// TIA Portal project "1200_SQL" (V16)

(* hardware
DEVICE "S7-1200 station_1"  S7-1200 Station
   slot 0: "Rack_0"  S7-1200 Rack  Rack  V1.0
   slot 1: "PLC_1"  CPU 1215C DC/DC/Rly  6ES7 215-1HG40-0XB0  V4.4
*)

// ===== PLC "PLC_1"  CPU 1215C DC/DC/Rly =====

VAR_GLOBAL   // PLC tag table "Default tag table"
   "Tag_1" AT %M10.0 : Bool;
   "Tag_2" AT %M30.0 : Bool;
   "System_Byte" AT %MB1 : Byte;
   "FirstScan" AT %M1.0 : Bool;
   "DiagStatusUpdate" AT %M1.1 : Bool;
   "AlwaysTRUE" AT %M1.2 : Bool;
   "AlwaysFALSE" AT %M1.3 : Bool;
   "Clock_Byte" AT %MB0 : Byte;
   "Clock_10Hz" AT %M0.0 : Bool;
   "Clock_5Hz" AT %M0.1 : Bool;
   "Clock_2.5Hz" AT %M0.2 : Bool;
   "Clock_2Hz" AT %M0.3 : Bool;
   "Clock_1.25Hz" AT %M0.4 : Bool;
   "Clock_1Hz" AT %M0.5 : Bool;
   "Clock_0.625Hz" AT %M0.6 : Bool;
   "Clock_0.5Hz" AT %M0.7 : Bool;
   "Tag_3" AT %M1000.0 : Bool;
   "Tag_4" AT %M1000.1 : Bool;
   "Tag_5" AT %M1000.2 : Bool;
   "Tag_6" AT %M29.0 : Bool;
   "Tag_7" AT %M1000.5 : Bool;
END_VAR

TYPE "typeUseCaseSpecificTokenRow"
   STRUCT
      length : Byte;
      data : DWord;
   END_STRUCT;
END_TYPE

TYPE "typeUseCaseSpecificData"
   STRUCT
      header : "LSql_typeTDSPacketHeader";   // TDS Protocol header
      tokenColumnMetaData : Array[0..23] of Byte;   // information about the columns returned in the tokenRows - depends on user data
      tokenRows : Array[0..14] of "typeUseCaseSpecificTokenRow";   // Rows returned for the SQL Batch - sturcture depends on user data!
      bytes : Array[0..867] of Byte;
   END_STRUCT;
   // // header."type" : type of TDS package (4 = Server Response)
   // // header.status : status of the TDS package (1= last package, 0 = more packages follow)
   // // header.length : length of the TDS response
   // // header.SPID : process id of the SQL server
   // // header.PacketID : id of one message for a paket
   // // header.Window : not used - should be ignored by user
END_TYPE

// folder: LSql

TYPE "LSql_typeDiagnostics"
TITLE = typeDiagnosticsTemplate
   STRUCT
      status : Word;   // Status of the Block or error identification when error occurred
      subfunctionStatus : Word;   // Status or return value of called FB's, FCs and system blocks
      stateNumber : DInt;   // State in the state machine of the block where the error occurred
   END_STRUCT;
END_TYPE

TYPE "LSql_typeLoginInformation"
   STRUCT
      hostName : String;   // optional: name of local host
      userName : String;   // mandatory: username for login to database
      password : String;   // mandatory: password for login to database
      appName : String;   // optional: name of app connectiong to database
      serverName : String;   // mandatory: servername of database
      libraryName : String;   // optional: name of ui
      local : String;   // optional: language used in ui
      databaseName : String;   // mandatory: database to read or write from
      sspi : String;   // optional / not supported: encryption via sspi
      attachDbfile : String;   // optional: filename to add at transfer
      changePassword : String;   // optional: new password if old one shold be changed
   END_STRUCT;
END_TYPE

TYPE "LSql_typeConnectionSettings"
   STRUCT
      interfaceSettings : TCON_IP_v4;
      loginInformation : "LSql_typeLoginInformation";
   END_STRUCT;
END_TYPE

// folder: LSql/Helpers

TYPE "LSql_typeTDSPacketHeader"
   STRUCT
      "type" : Byte;
      status : Byte;
      length : UInt;
      SPID : Word;
      PacketID : Byte;
      Window : Byte;
   END_STRUCT;
END_TYPE

TYPE "LSql_typeLoginData"
   STRUCT
      header : Struct   // general tds header / properties of the TDS message
         "type" : Byte := 16#10;   // fixed value for login / permanent value depending on message type (16#01: SQL-Batch, 16#10: Login, 16#12: PreLogin)
         status : Byte := 16#01;   // statusflags / message status
         length : Word := 16#0090;   // size including packet header (header + login7) / message length ( = header + login data )
         spid : Word := 16#0000;   // process id on the server (for debuging)
         packet : Byte := 16#01;   // packet number for identify messages (with messages more than one packet) / packet number (used to set together message from serveral others)
         window : Byte := 16#00;   // not used / not used - must be set to 16#00
      END_STRUCT;
      login : Struct   // login message
         length : DWord := 16#88000000;   // length of the login / length of the login message
         tdsVersion : DWord := 16#02000972;   // tds version / TDS version
         packetSize : DWord := 16#00100000;   // packet size requested by the client / requested package size
         clientProgVer : DWord := 16#00000007;   // version of the interface being used by the client / interface version of the client
         clientId : DWord := 16#00010000;   // client ID / client id
         conncetionId : DWord := 16#00000000;   // connection ID (used with "always up" backup servers) / connection id - used for permanent connections
         optionFlags1 : Byte := 16#E0;   // optionFlags1 (fByteOrder, fChar, fFloat(2), fDumpLoad, fUseDB, fDatabasem fSetLang) / settings 1
         optionFlags2 : Byte := 16#03;   // optionFlags2 (fLanguage, fODBC, fTransBoundary, fCacheConnect, fUserType(2), fIntSecurity) / settings 2
         typeFlags : Byte := 16#00;   // typeFlags (fSQLType, fOLEDB, fReadOnlyIntent)
         optionFlags3 : Byte := 16#00;   // optionFlags3 (fChangePassword, fSendYukonBinaryXML, fUserInstance, fUnknownCollationHandling, fExtensions) / settings 3
         clientTimeZone : DWord := 16#E0010000;   // time zone / timezone of the client
         clientLCID : DWord := 16#09040000;   // language code identifier / language id
         offsetLength : Struct   // information where the data is located in the data stream / offest and length of information in message
            hostName : Struct   // client machine name / local hostname ( not mandatory )
               offset : Word := 16#5E00;   // offset in bytes relative to the message start (ibHostName) / offset in bytes to beginning of the header
               length : Word := 16#0800;   // message length in bytes (cchHostName) / length of the hostname, including zero bytes
            END_STRUCT;
            userName : Struct   // client user ID / user name to log on to server ( mandatory )
               offset : Word := 16#6E00;   // offset in bytes relative to the message start (ibUserName) / offset in bytes to beginning of the header
               length : Word := 16#0200;   // message length in bytes (cchUserName) / length of the user name, including zero bytes
            END_STRUCT;
            password : Struct   // password / password to the corresponding user name
               offset : Word := 16#7200;   // offset in bytes relative to the message start (ibPassword) / offset in bytes to beginning of the header
               length : Word := 16#0000;   // message length in bytes (cchPassword) / length of the password, including zero bytes
            END_STRUCT;
            appName : Struct   // client application name / name of the app that has to access the server ( not mandatory )
               offset : Word := 16#7200;   // offset in bytes relative to the message start (ibAppName) / offset in bytes to beginning of the header
               length : Word := 16#0700;   // message length in bytes (cchAppName) / length of the app name, including zero bytes
            END_STRUCT;
            serverName : Struct   // server name / name of the server to establish connection to ( mandatory )
               offset : Word := 16#8000;   // offset in bytes relative to the message start (ibServerName) / offset in bytes to beginning of the header
               length : Word := 16#0000;   // message length in bytes (cchServerName) / length of the server name, including zero bytes
            END_STRUCT;
            unused : Struct   // reserved until TDS 7.4 / currently not used - must be contained in login message
               offset : Word := 16#8000;   // offset in bytes relative to the message start (ibUnused)
               length : Word := 16#0000;   // message length in bytes (cchUnused)
            END_STRUCT;
            libraryName : Struct   // interface library name (i.e ODBC or OLEDB) / name of the user interface ( not mandatory )
               offset : Word := 16#8000;   // offset in bytes relative to the message start (ibCltIntName) / offset in bytes to beginning of the header
               length : Word := 16#0400;   // message length in bytes (cchCltIntName) / length of the user interface name, including zero bytes
            END_STRUCT;
            local : Struct   // initial language / language used for communication ( not mandatory )
               offset : Word := 16#8800;   // offset in bytes relative to the message start (ibLanguage) / offset in bytes to beginning of the header
               length : Word := 16#0000;   // message length in bytes (cchLanguage) / length of the language, including zero bytes
            END_STRUCT;
            databaseName : Struct   // inital database(overrides the user ID's default database) / database to changed or read ( mandatory )
               offset : Word := 16#8800;   // offset in bytes relative to the message start (ibDatabase) / offset in bytes to beginning of the header
               length : Word := 16#0000;   // message length in bytes (cchDatabase) / length of the database name, including zero bytes
            END_STRUCT;
            clientId : Array[0..5] of Byte;   // MAC adress
            sspi : Struct   // sspi data / Encryption via SSPI. not mandatory, not supported
               offset : Word := 16#8800;   // offset in bytes relative to the message start (ibSspi) / offset in bytes to beginning of the header
               length : Word := 16#0000;   // message length in bytes (cchSspi) / length of the sspi, including zero bytes
            END_STRUCT;
            atchDbFile : Struct   // file name for a database that is to be attached during the connection process / file name to be attached during connection setup
               offset : Word := 16#8800;   // offset in bytes relative to the message start / offset in bytes to beginning of the header
               length : Word := 16#0000;   // message length in bytes / length of the file name, including zero bytes
            END_STRUCT;
            changePassword : Struct   // new password for the specified login / new password, when old password should be changed ( not mandatory for login )
               offset : Word := 16#8800;   // offset in bytes relative to the message start / offset in bytes to beginning of the header
               length : Word := 16#0000;   // message length in bytes / length of the new password, including zero bytes
            END_STRUCT;
            cbSspiLong : DWord := 16#00000000;   // used for long sspi data / used for large sbsspi data
         END_STRUCT;
         data : Array[0..1023] of Byte;   // loginData / area used for login information
      END_STRUCT;
   END_STRUCT;
   // login.offsetLength.clientId[0] := 16#0D;
   // login.offsetLength.clientId[1] := 16#7D;
   // login.offsetLength.clientId[2] := 16#95;
   // login.offsetLength.clientId[3] := 16#36;
   // login.offsetLength.clientId[4] := 16#63;
   // login.offsetLength.clientId[5] := 16#28;
END_TYPE

TYPE "LSql_typePreloginData"
   STRUCT
      header : Struct   // general tds header / properties of TDS message
         "type" : Byte := 16#12;   // fixed value for preLogin / numeric values for type of mesage (16#01: SQL-Batch, 16#10: Login, 16#12: PreLogin)
         status : Byte := 16#01;   // status flags / status flag of the message
         length : Word := 16#005E;   // size including packet header (header + preLoginMessage) / length of message ( header + prelogin )
         channel : Word := 16#0000;   // process id on the server (for debuging) / process id on the server
         packet : Byte := 16#01;   // packet number for identify messages (with messages more than one packet) / packet number (used to set together message from serveral others)
         window : Byte := 16#00;   // not used / not used - must be set to 16#00
      END_STRUCT;
      data : Struct   // prelogin message / preLogin message
         option : Struct   // information where the data is located in the data stream / offset and length of information contained in message
            "version" : Struct   // version of the sender / version of sender
               token : Byte := 16#00;   // fixed value for version token / permanent value for version
               offset : Word := 16#0024;   // offset in bytes relative to the message start / offset in bytes - relative to beginning of header
               length : Word := 16#0006;   // message length in bytes / message length
            END_STRUCT;
            encryption : Struct   // encryption settings / encryption of message
               token : Byte := 16#01;   // fixed value for encryption token / permanent value for encryption
               offset : Word := 16#002A;   // offset in bytes relative to the message start / offset in bytes - relative to beginning of header
               length : Word := 16#0001;   // message length in bytes / message length
            END_STRUCT;
            instOpt : Struct   // instOpt (name of the database or just 16#00) / name of the database
               token : Byte := 16#02;   // fixed value for instOpt token / permanent value
               offset : Word := 16#002B;   // offset in bytes relative to the message start / offset in bytes - relative to beginning of header
               length : Word := 16#0001;   // message length in bytes / message length
            END_STRUCT;
            threadId : Struct   // client application threadId (used for debugging purposes) / user thread id
               token : Byte := 16#03;   // fixed value for thread Id token / permanent value for thread id
               offset : Word := 16#002C;   // offset in bytes relative to the message start / offset in bytes - relative to beginning of header
               length : Word := 16#0004;   // message length in bytes / message length
            END_STRUCT;
            mars : Struct   // mars settings / not used - allows sending and execution of several messages at the same time
               token : Byte := 16#04;   // fixed value for mars token / permanent value for mars
               offset : Word := 16#0030;   // offset in bytes relative to the message start / offset in bytes - relative to beginning of header
               length : Word := 16#0001;   // message length in bytes / message length
            END_STRUCT;
            traceId : Struct   // client application traceId (used for debugging purposes) / user trace id
               token : Byte := 16#05;   // fixed value for traceId token / permanent value for trace id
               offset : Word := 16#0031;   // offset in bytes relative to the message start / offset in bytes - relative to beginning of header
               length : Word := 16#0024;   // message length in bytes / message length
            END_STRUCT;
            fedAuthRequired : Struct   // authentification library requirement when using Integrated Authentification identity / authentication request
               token : Byte := 16#06;   // fixed value for fedAuthRequired token / permanent value for fedAuthRequired
               offset : Word := 16#0055;   // offset in bytes relative to the message start / offset in bytes - relative to beginning of header
               length : Word := 16#0001;   // message length in bytes / message length
            END_STRUCT;
            terminator : Byte := 16#FF;   // fixed value for end of option / permanent value for terminator
         END_STRUCT;
         data : Array[0..49] of Byte;   // message data bytes / content of message
      END_STRUCT;
   END_STRUCT;
   // data.data[0] := 16#0C;   // version (12.0)
   // data.data[1] := 16#00;   // version (12.0)
   // data.data[2] := 16#13;   // subbuild (5000)
   // data.data[3] := 16#88;   // subbuild (5000)
   // data.data[4] := 16#00;   // subbuild (5000)
   // data.data[5] := 16#00;   // subbuild (5000)
   // data.data[6] := 16#02;   // encryption off
   // data.data[7] := 16#00;   // instOpt
   // data.data[8] := 16#00;   // thread ID
   // data.data[9] := 16#00;   // thread ID
   // data.data[10] := 16#B8;   // thread ID
   // data.data[11] := 16#0D;   // thread ID
   // data.data[12] := 16#00;   // mars (0 =off)
   // data.data[13] := 16#DD;   // traceId
   // data.data[14] := 16#DA;   // traceId
   // data.data[15] := 16#47;   // traceId
   // data.data[16] := 16#1C;   // traceId
   // data.data[17] := 16#6C;   // traceId
   // data.data[18] := 16#79;   // traceId
   // data.data[19] := 16#D4;   // traceId
   // data.data[20] := 16#4D;   // traceId
   // data.data[21] := 16#AC;   // traceId
   // data.data[22] := 16#52;   // traceId
   // data.data[23] := 16#7F;   // traceId
   // data.data[24] := 16#33;   // traceId
   // data.data[25] := 16#86;   // traceId
   // data.data[26] := 16#C7;   // traceId
   // data.data[27] := 16#42;   // traceId
   // data.data[28] := 16#6A;   // traceId
   // data.data[29] := 16#BB;   // traceId
   // data.data[30] := 16#F2;   // traceId
   // data.data[31] := 16#26;   // traceId
   // data.data[32] := 16#EF;   // traceId
   // data.data[33] := 16#11;   // traceId
   // data.data[34] := 16#72;   // traceId
   // data.data[35] := 16#0C;   // traceId
   // data.data[36] := 16#48;   // traceId
   // data.data[37] := 16#A8;   // traceId
   // data.data[38] := 16#66;   // traceId
   // data.data[39] := 16#4B;   // traceId
   // data.data[40] := 16#F4;   // traceId
   // data.data[41] := 16#4A;   // traceId
   // data.data[42] := 16#CD;   // traceId
   // data.data[43] := 16#E2;   // traceId
   // data.data[44] := 16#A4;   // traceId
   // data.data[45] := 16#01;   // traceId
   // data.data[46] := 16#00;   // traceId
   // data.data[47] := 16#00;   // traceId
   // data.data[48] := 16#00;   // traceId
   // data.data[49] := 16#01;   // fedAuthRequirement
END_TYPE

TYPE "LSql_typeSqlBatchData"
   STRUCT
      header : Struct   // general tds header / properties of the TDS message
         "type" : Byte := 16#01;   // fixed value for preLogin / permanent value depending on message type (16#01: SQL-Batch, 16#10: Login, 16#12: PreLogin)
         status : Byte := 16#01;   // status flags / message status
         length : Word := 16#001E;   // size including packet header (header + preLoginMessage) / message length ( = header + login data )
         channel : Word := 16#0000;   // process id on the server (for debuging) / process id on the server
         packet : Byte := 16#01;   // packet number for identify messages (with messages more than one packet) / packet number (used to set together message from serveral others)
         window : Byte := 16#00;   // not used / not used - must be set to 16#00
      END_STRUCT;
      sqlBatch : Struct   // sqlBatch message
         totalLength : DWord := 16#16000000;   // fixed value for total length (totalLength + header) / length of sqlBatch without SQL-text
         header : Struct   // sqlBatch header / settings in header
            headerLength : DWord := 16#12000000;   // fixed value for header length / length of the header
            headerType : Word := 16#0200;   // fixed value for sqlBatch header / type of the header
            mars : Struct   // settings for mars / parameters for mars, not relevant
               transactionDescriptor : Array[0..7] of Byte;   // pritority / description of the transaction
               outstandingRequestCount : DWord := 16#01000000;   // request number / ascending numbering of the incoming requests
            END_STRUCT;
         END_STRUCT;
         sqlText : Array[0..1023] of Byte;   // SQL-command as string / area for sql command
      END_STRUCT;
   END_STRUCT;
END_TYPE

TYPE "LSql_typePacketDataQueryResponse"
   STRUCT
      columns : Word;
      usertype : DWord;
      flags : Word;
      "type" : Byte;
      typeSize : Byte;
      colNameLength : Byte;
      columns_1 : Array[0..7] of Byte;
      row_tokens : Array[0..100] of "typeUseCaseSpecificTokenRow";
   END_STRUCT;
END_TYPE

// folder: (top level)

DATA_BLOCK "SqlConfig"   // DB2
{ S7_Optimized_Access := 'TRUE' }
VERSION : 0.1
   VAR
      connectionSettings : "LSql_typeConnectionSettings";
      enableLSql : Bool := true;   // enables LSql block (starts connection and login, waits for execute commands)
      diagnostics : "LSql_typeDiagnostics";
      executeSqlCommand : Bool;   // trigger to execute a single sql command. EnableLSql must be true before triggering
   END_VAR
BEGIN
   connectionSettings.interfaceSettings.InterfaceId := 64;
   connectionSettings.interfaceSettings.ID := 16#10;
   connectionSettings.interfaceSettings.ActiveEstablished := true;
   connectionSettings.interfaceSettings.RemoteAddress.ADDR[2] := 168;
   connectionSettings.interfaceSettings.RemoteAddress.ADDR[3] := 0;
   connectionSettings.interfaceSettings.RemoteAddress.ADDR[4] := 100;
   connectionSettings.interfaceSettings.RemotePort := 1433;
   connectionSettings.loginInformation.userName := 'sa';
   connectionSettings.loginInformation.password := '12345';
   connectionSettings.loginInformation.appName := '';
   connectionSettings.loginInformation.serverName := 'SQLExpress';
   connectionSettings.loginInformation.databaseName := 'PLC_S71200';
   connectionSettings.interfaceSettings.RemoteAddress.ADDR[1] := 192;
END_DATA_BLOCK

DATA_BLOCK "SqlCommands"   // DB3
{ S7_Optimized_Access := 'TRUE' }
VERSION : 0.1
   VAR
      sqlCommandsInsert : Array[0..6] of String;
   END_VAR
BEGIN
   sqlCommandsInsert[0] := 'INSERT INTO tb_mirrorPlcL1 VALUES (7,8, 9)';
   sqlCommandsInsert[1] := 'UPDATE tb_mirrorPlcL1 SET timeStop = 1111, qtStop = 2222 WHERE workstation_id = 1';
   sqlCommandsInsert[2] := 'SELECT workstation_id FROM tb_mirrorPlcL1';
   sqlCommandsInsert[3] := 'SELECT Amount FROM PLCDATA_2 WHERE Fruit = $'Apple$'';
   sqlCommandsInsert[4] := 'Select Fruit from PLCDATA_2 where color = $'red$'';
   sqlCommandsInsert[5] := 'insert into PLCDATA_3 values (7, $'2020-01-01 10:23:24.125$')';
END_DATA_BLOCK

DATA_BLOCK "SqlReceive"   // DB8
{ S7_Optimized_Access := 'TRUE' }
VERSION : 0.1
   VAR
      data : "typeUseCaseSpecificData";
   END_VAR
BEGIN
END_DATA_BLOCK

DATA_BLOCK "DBRecordDatasSQL"   // DB10
{ S7_Optimized_Access := 'TRUE' }
VERSION : 0.1
   VAR
      StrStartSQL : String := 'UPDATE tb_mirrorPlcL1 SET  timeStop=';   // SQL command
      SQLValueCol1 : String := '';   // Data part 1
      SQLColumn2 : String := 'qtStop=';
      SQLValueCol2 : String := '';   // Data part 2
      SQLWhere : String := ' WHERE workstation_id=';
      SQLComma : String := ', ';
      SQLBrakeRight : String := ')';
      SQLFullCommandW1 : String;   // Joint command, part1 and part2
      Station1_T1 : Array[0..7] of Char;
   END_VAR
BEGIN
   Station1_T1[7] := '0';
   Station1_T1[6] := '0';
   Station1_T1[5] := '0';
   Station1_T1[4] := '0';
   Station1_T1[3] := '0';
   Station1_T1[2] := '0';
   Station1_T1[1] := '0';
   Station1_T1[0] := '0';
END_DATA_BLOCK

// folder: LSql

DATA_BLOCK "InstLSql_Microsoft"   // DB1
{ S7_Optimized_Access := 'TRUE' }
AUTHOR : (department/personInCharge/contact)
FAMILY : (family)
VERSION : 0.1
// stored: InstanceOfName LSql_Microsoft
"LSql_Microsoft"
BEGIN
END_DATA_BLOCK

// folder: (top level)

FUNCTION "RecordDatasSQL" : Void   // FC10, LAD
{ S7_Optimized_Access := 'TRUE' }
VERSION : 0.1
   VAR_TEMP   // added for the SCL form of the ladder/FBD networks
      _w1 : Bool;
      _w2 : Bool;
      _w3 : Bool;
      _w4 : Bool;
   END_VAR
BEGIN

REGION Network 1
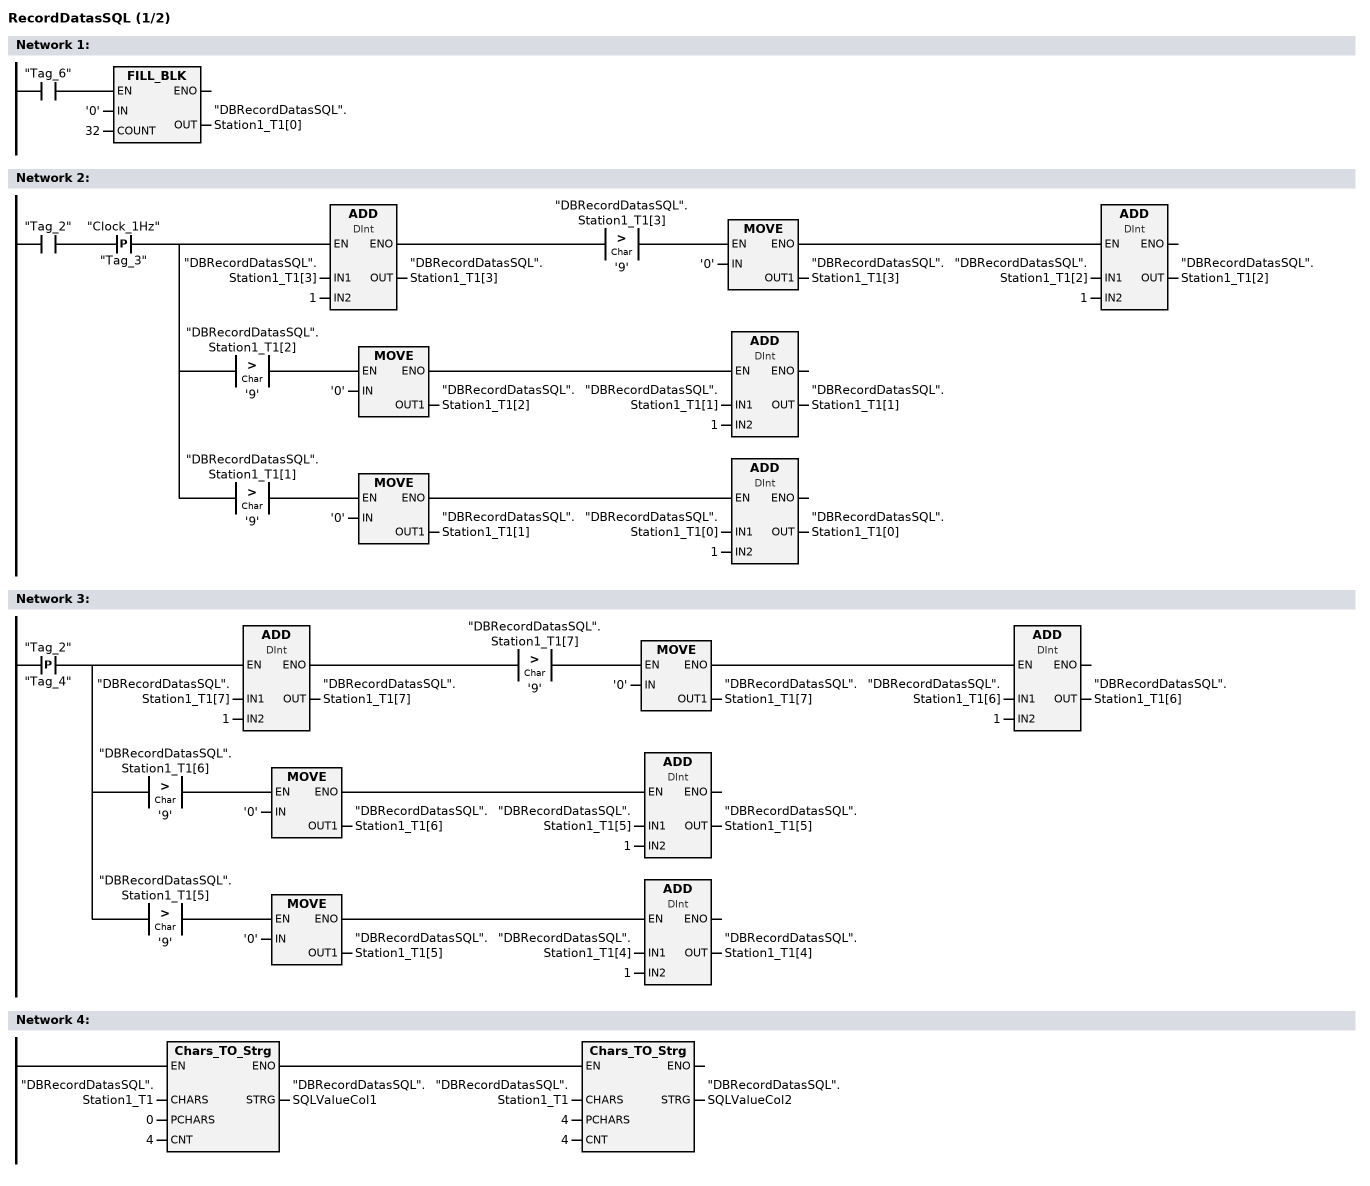
   RUNG wire#powerrail
      Contact( "Tag_6" )
      FillBlockI(in := '0', count := 32, out => "DBRecordDatasSQL".Station1_T1[0])
   END_RUNG
   // the same network as SCL:
   IF "Tag_6" THEN FILL_BLK(IN := '0', COUNT := 32, OUT => "DBRecordDatasSQL".Station1_T1[0]); END_IF;
END_REGION

REGION Network 2
   RUNG wire#powerrail
      Contact( "Tag_2" )
      P_Contact(operand := "Clock_1Hz", bit := "Tag_3")
      wire#w1
      { S7_Templates := "SrcType := DInt" } Add(in1 := "DBRecordDatasSQL".Station1_T1[3], in2 := 1, out => "DBRecordDatasSQL".Station1_T1[3])
      { S7_Templates := "SrcType := Char" } GT_Contact(in1 := "DBRecordDatasSQL".Station1_T1[3], in2 := '9')
      Move(in := '0', out1 => "DBRecordDatasSQL".Station1_T1[3])
      { S7_Templates := "SrcType := DInt" } Add(in1 := "DBRecordDatasSQL".Station1_T1[2], in2 := 1, out => "DBRecordDatasSQL".Station1_T1[2])
   END_RUNG
   RUNG wire#w1
      { S7_Templates := "SrcType := Char" } GT_Contact(in1 := "DBRecordDatasSQL".Station1_T1[2], in2 := '9')
      Move(in := '0', out1 => "DBRecordDatasSQL".Station1_T1[2])
      { S7_Templates := "SrcType := DInt" } Add(in1 := "DBRecordDatasSQL".Station1_T1[1], in2 := 1, out => "DBRecordDatasSQL".Station1_T1[1])
   END_RUNG
   RUNG wire#w1
      { S7_Templates := "SrcType := Char" } GT_Contact(in1 := "DBRecordDatasSQL".Station1_T1[1], in2 := '9')
      Move(in := '0', out1 => "DBRecordDatasSQL".Station1_T1[1])
      { S7_Templates := "SrcType := DInt" } Add(in1 := "DBRecordDatasSQL".Station1_T1[0], in2 := 1, out => "DBRecordDatasSQL".Station1_T1[0])
   END_RUNG
   // the same network as SCL:
   #_w1 := "Tag_2" AND "Clock_1Hz" AND NOT "Tag_3";   // rising edge of "Clock_1Hz"
   "Tag_3" := "Clock_1Hz";
   IF #_w1 THEN "DBRecordDatasSQL".Station1_T1[3] := "DBRecordDatasSQL".Station1_T1[3] + 1; END_IF;
   #_w2 := #_w1 AND ("DBRecordDatasSQL".Station1_T1[3] > '9');
   IF #_w2 THEN
       "DBRecordDatasSQL".Station1_T1[3] := '0';
       "DBRecordDatasSQL".Station1_T1[2] := "DBRecordDatasSQL".Station1_T1[2] + 1;
   END_IF;
   #_w3 := #_w1 AND ("DBRecordDatasSQL".Station1_T1[2] > '9');
   IF #_w3 THEN
       "DBRecordDatasSQL".Station1_T1[2] := '0';
       "DBRecordDatasSQL".Station1_T1[1] := "DBRecordDatasSQL".Station1_T1[1] + 1;
   END_IF;
   #_w4 := #_w1 AND ("DBRecordDatasSQL".Station1_T1[1] > '9');
   IF #_w4 THEN
       "DBRecordDatasSQL".Station1_T1[1] := '0';
       "DBRecordDatasSQL".Station1_T1[0] := "DBRecordDatasSQL".Station1_T1[0] + 1;
   END_IF;
END_REGION

REGION Network 3
   RUNG wire#powerrail
      P_Contact(operand := "Tag_2", bit := "Tag_4")
      wire#w1
      { S7_Templates := "SrcType := DInt" } Add(in1 := "DBRecordDatasSQL".Station1_T1[7], in2 := 1, out => "DBRecordDatasSQL".Station1_T1[7])
      { S7_Templates := "SrcType := Char" } GT_Contact(in1 := "DBRecordDatasSQL".Station1_T1[7], in2 := '9')
      Move(in := '0', out1 => "DBRecordDatasSQL".Station1_T1[7])
      { S7_Templates := "SrcType := DInt" } Add(in1 := "DBRecordDatasSQL".Station1_T1[6], in2 := 1, out => "DBRecordDatasSQL".Station1_T1[6])
   END_RUNG
   RUNG wire#w1
      { S7_Templates := "SrcType := Char" } GT_Contact(in1 := "DBRecordDatasSQL".Station1_T1[6], in2 := '9')
      Move(in := '0', out1 => "DBRecordDatasSQL".Station1_T1[6])
      { S7_Templates := "SrcType := DInt" } Add(in1 := "DBRecordDatasSQL".Station1_T1[5], in2 := 1, out => "DBRecordDatasSQL".Station1_T1[5])
   END_RUNG
   RUNG wire#w1
      { S7_Templates := "SrcType := Char" } GT_Contact(in1 := "DBRecordDatasSQL".Station1_T1[5], in2 := '9')
      Move(in := '0', out1 => "DBRecordDatasSQL".Station1_T1[5])
      { S7_Templates := "SrcType := DInt" } Add(in1 := "DBRecordDatasSQL".Station1_T1[4], in2 := 1, out => "DBRecordDatasSQL".Station1_T1[4])
   END_RUNG
   // the same network as SCL:
   #_w1 := "Tag_2" AND NOT "Tag_4";   // rising edge of "Tag_2"
   "Tag_4" := "Tag_2";
   IF #_w1 THEN "DBRecordDatasSQL".Station1_T1[7] := "DBRecordDatasSQL".Station1_T1[7] + 1; END_IF;
   #_w2 := #_w1 AND ("DBRecordDatasSQL".Station1_T1[7] > '9');
   IF #_w2 THEN
       "DBRecordDatasSQL".Station1_T1[7] := '0';
       "DBRecordDatasSQL".Station1_T1[6] := "DBRecordDatasSQL".Station1_T1[6] + 1;
   END_IF;
   #_w3 := #_w1 AND ("DBRecordDatasSQL".Station1_T1[6] > '9');
   IF #_w3 THEN
       "DBRecordDatasSQL".Station1_T1[6] := '0';
       "DBRecordDatasSQL".Station1_T1[5] := "DBRecordDatasSQL".Station1_T1[5] + 1;
   END_IF;
   #_w4 := #_w1 AND ("DBRecordDatasSQL".Station1_T1[5] > '9');
   IF #_w4 THEN
       "DBRecordDatasSQL".Station1_T1[5] := '0';
       "DBRecordDatasSQL".Station1_T1[4] := "DBRecordDatasSQL".Station1_T1[4] + 1;
   END_IF;
END_REGION

REGION Network 4
   // no SCL statement known for Chars_TO_Strg: written as a call
   // ENO of a box is taken as its EN; it also drops when the box reports an error
   Chars_TO_Strg(Chars := "DBRecordDatasSQL".Station1_T1,
                 pChars := 0,
                 Cnt := 4,
                 Strg => "DBRecordDatasSQL".SQLValueCol1);
   Chars_TO_Strg(Chars := "DBRecordDatasSQL".Station1_T1,
                 pChars := 4,
                 Cnt := 4,
                 Strg => "DBRecordDatasSQL".SQLValueCol2);
END_REGION

REGION Network 5: PartA String
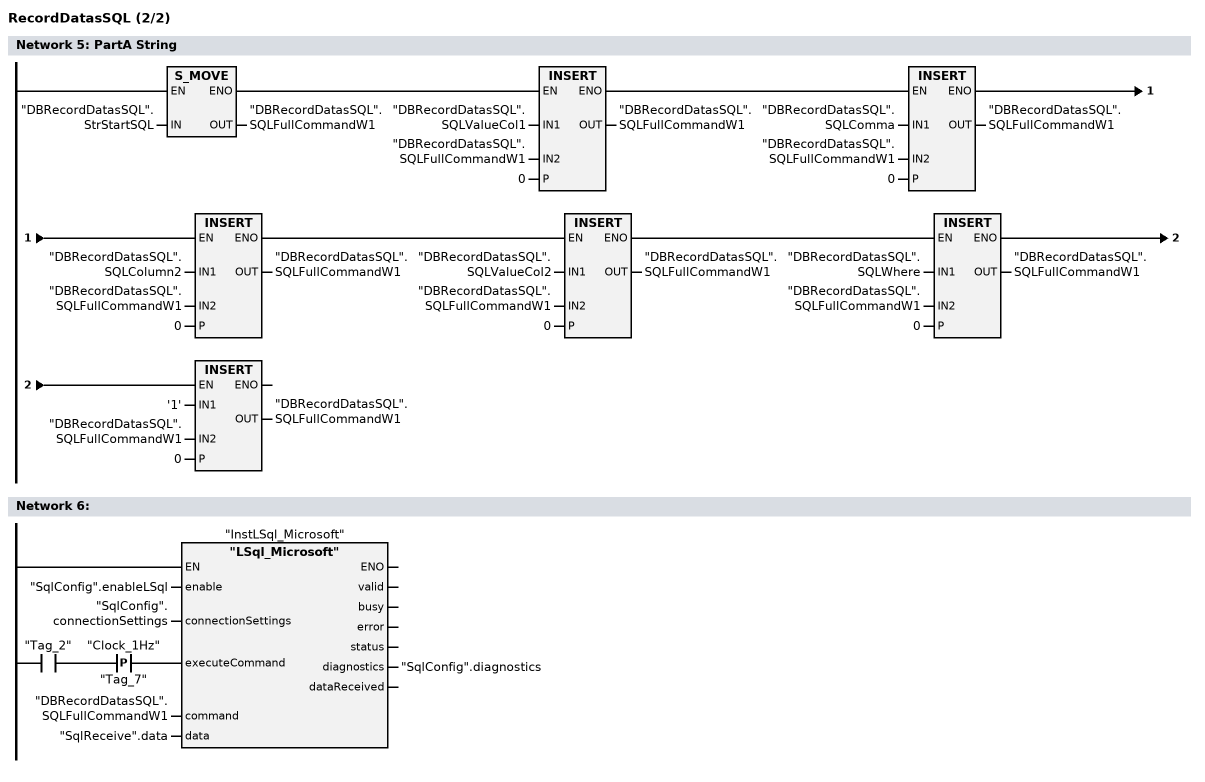
   "DBRecordDatasSQL".SQLFullCommandW1 := "DBRecordDatasSQL".StrStartSQL;
   "DBRecordDatasSQL".SQLFullCommandW1 := INSERT(IN1 := "DBRecordDatasSQL".SQLValueCol1,
                           IN2 := "DBRecordDatasSQL".SQLFullCommandW1,
                           P := 0);
   "DBRecordDatasSQL".SQLFullCommandW1 := INSERT(IN1 := "DBRecordDatasSQL".SQLComma,
                           IN2 := "DBRecordDatasSQL".SQLFullCommandW1,
                           P := 0);
   "DBRecordDatasSQL".SQLFullCommandW1 := INSERT(IN1 := "DBRecordDatasSQL".SQLColumn2,
                           IN2 := "DBRecordDatasSQL".SQLFullCommandW1,
                           P := 0);
   "DBRecordDatasSQL".SQLFullCommandW1 := INSERT(IN1 := "DBRecordDatasSQL".SQLValueCol2,
                           IN2 := "DBRecordDatasSQL".SQLFullCommandW1,
                           P := 0);
   "DBRecordDatasSQL".SQLFullCommandW1 := INSERT(IN1 := "DBRecordDatasSQL".SQLWhere,
                           IN2 := "DBRecordDatasSQL".SQLFullCommandW1,
                           P := 0);
   "DBRecordDatasSQL".SQLFullCommandW1 := INSERT(IN1 := '1', IN2 := "DBRecordDatasSQL".SQLFullCommandW1, P := 0);
END_REGION

REGION Network 6
   RUNG wire#powerrail
      "InstLSql_Microsoft"(executeCommand := wire#w1, enable := "SqlConfig".enableLSql, connectionSettings := "SqlConfig".connectionSettings, command := "DBRecordDatasSQL".SQLFullCommandW1, data := "SqlReceive".data, valid =>, busy =>, error =>, status =>, diagnostics => "SqlConfig".diagnostics, dataReceived =>)
   END_RUNG
   RUNG wire#powerrail
      Contact( "Tag_2" )
      P_Contact(operand := "Clock_1Hz", bit := "Tag_7")
   END_RUNG wire#w1
   // the same network as SCL:
   #_w1 := "Tag_2" AND "Clock_1Hz" AND NOT "Tag_7";   // rising edge of "Clock_1Hz"
   "Tag_7" := "Clock_1Hz";
   "InstLSql_Microsoft"(enable := "SqlConfig".enableLSql,   // "LSql_Microsoft"
                        connectionSettings := "SqlConfig".connectionSettings,
                        executeCommand := #_w1,
                        command := "DBRecordDatasSQL".SQLFullCommandW1,
                        data := "SqlReceive".data,
                        diagnostics => "SqlConfig".diagnostics);
END_REGION
END_FUNCTION

ORGANIZATION_BLOCK "Main"   // OB1, LAD, ProgramCycle
TITLE = "Main Program Sweep (Cycle)"
{ S7_Optimized_Access := 'TRUE' }
VERSION : 0.1
   VAR_INPUT
      Initial_Call : Bool;   // Initial call of this OB
      Remanence : Bool;   // =True, if remanent data are available
   END_VAR
BEGIN

REGION Network 2
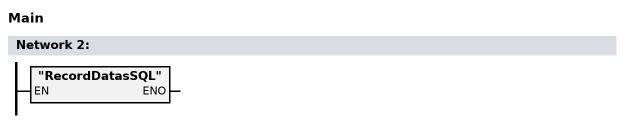
   RUNG wire#powerrail
      "RecordDatasSQL"()
   END_RUNG
   // the same network as SCL:
   "RecordDatasSQL"();
END_REGION
END_ORGANIZATION_BLOCK

// folder: LSql

FUNCTION_BLOCK "LSql_Microsoft"   // FB2, SCL
TITLE = Enable Template
{ S7_Optimized_Access := 'TRUE' }
AUTHOR : (department/personInCharge/contact)
FAMILY : (family)
VERSION : 0.1
// Template for an FB with Enable / Valid handling based on PLCopen standard "Function Blocks for Motion Control" V2.0
   VAR_INPUT
      enable : Bool;   // TRUE: Enable functionality of FB
      connectionSettings : "LSql_typeConnectionSettings";
      executeCommand : Bool;   // TRUE: execute sql command once
      command : String;   // SQL command to execute when executeSqlBatch = TRUE
   END_VAR
   VAR_OUTPUT
      valid : Bool;   // TRUE: Valid set of output values available at the FB
      busy : Bool;   // TRUE: FB is not finished and new output values can be expected
      error : Bool;   // TRUE: An error occurred during the execution of the FB
      status : Word := 16#7000;   // 16#0000 - 16#7FFF: Status of the FB, 16#8000 - 16#FFFF: Error identification
      diagnostics : "LSql_typeDiagnostics";   // Diagnostics information of FB (optional)
      dataReceived : Bool;   // TRUE: new data was received
   END_VAR
   VAR_IN_OUT
      data : "typeUseCaseSpecificData";   // response recieved from SQL server
   END_VAR
   VAR
      statEnableOld : Bool;   // Old value of 'enable' input for edge detection
      statEnable : Bool;   // current value of enable
      statValid : Bool;   // Static value for output 'valid'
      statBusy : Bool;   // Static value for output 'busy'
      statError : Bool;   // Static value for output 'error'
      statErrorUserCleared : Bool;   // Error occurred that can only be solved by user; rising edge at enable input necessary
      statErrorAutoCleared : Bool;   // Error occurred that can be acknowledged by FB
      statStatus : Word := 16#7000;   // Static value for output 'status'
      statSubfunctionStatus : Word;   // Status or return value of called FBs, FCs and system blocks
      statFBErrorState : DInt;   // State in the state machine of the block where the error occurred
      statFBState : DInt := 0;   // State in the state machine of the FB
      statDisablingCompleted : Bool;   // TRUE: Disabling has been completed
      statEmptyDiagnostics : "LSql_typeDiagnostics";   // Empty diagnostics information (for initialization purposes only)
      statReceivedBytes : UDInt;   // amount of data received from SQL server
      statExecuteSqlBatchOld : Bool;   // old value of 'executeSqlBatch' input
      statSqlBatchData : "LSql_typeSqlBatchData";   // sql batch data is copied here and length of data
      statSqlBatch : Array[0..2047] of Byte;   // sql batch data is inserted here as word
      statSqlBatchLen : DInt;   // length of sql batch data
      statWriter : Int;   // write length of data to DB
      statStatusSqlBatchIntToWord : Word;   // output of Int_to_word for SqlBatch command
      statLoginData : "LSql_typeLoginData";   // sql login data is copied here and length of data
      statLogin : Array[0..2047] of Byte;   // sql login data is inserted here as word
      statLoginLen : DInt;   // length of sql login data
      statStatusLoginIntToWord : Word;   // output of Int_to_word for Sql Login
      statStatusPreLoginIntToWord : Word;   // output of Int_to_word for Sql PreLogin
      statPreLogin : Array[0..2047] of Byte;   // sql prelogin data is inserted here as word
      statPreLoginLen : DInt;   // length of sql prelogin data
      statPreLoginCache : Array[0..2047] of Byte;   // sql prelogin data cache
      statPreLoginData : "LSql_typePreloginData";   // sql prelogin data is copied here and length of data
      instTsend : TSEND;   // instance for calling systemfunction Tsend
      instTcon : TCON;   // instance for calling systemfunction tcon
      instTrcv : TRCV;   // instance for calling systemfunction trcv
      instTdiscon : TDISCON;   // instance for calling systemfunction tdiscon
      statErrorWriteData : Bool;   // stat for output of WriteData in case of error
      statWriteData : Word;   // save output form WriteData
      statTransmissionSqlCommand : Bool;   // data stream for sql command was created, start tsend
      statSqlDataReceived : Bool;   // trcv got data from SQL server
   END_VAR
   VAR_TEMP
      tempPos : DInt;   // save position before writing data to byte array
      tempLength : Word;   // just necessary for running FC"writeData" / length of sql command data
      tempCounter : DInt;   // counter used for filling prelogin data from cache to byte array
      tempGaps : Int;   // count zero bytes in prelogin data
      tempLengthAsInt : DInt;   // save length as int after conversion
      tempLengthRor : DInt;   // save length after rotating to the right
   END_VAR
   VAR CONSTANT
      ERR_TDISCON_REMOTE_TERMINATION : Word := 16#80A3;   // Error: TDISCON, The connections is already terminated OR doesn't exist
      FB_STATE_NO_PROCESSING : DInt := 0;   // FB state: No processing
      FB_STATE_DISABLING : DInt := 1;   // FB state: Disconnect after enable input is set to false and deinitialize FBs
      FB_STATE_INITIAL_DISCON : DInt := 2;   // FB state: disconnect before initial connect
      FB_STATE_CONNECT : DInt := 3;   // FB state: Connect to database server
      FB_STATE_PRELOGIN : DInt := 4;   // FB state: Prelogin to Sql server
      FB_STATE_LOGIN : DInt := 5;   // FB state: Login to Sql server
      FB_STATE_SENDLOGIN : DInt := 6;   // FB state: send login data that was parsed in FB_STATE_LOGIN
      FB_STATE_SQLBATCH : DInt := 7;   // FB state: wait in this state for triggers of executeSqlBatch, archive packages from trcv
      STATUS_NO_CALL : Word := 16#7000;   // No job being currently processed
      STATUS_FIRST_CALL : Word := 16#7001;   // First call after incoming new job (rising edge 'enable')
      STATUS_SUBSEQUENT_CALL : Word := 16#7002;   // Subsequent call during active processing without further details
      STATUS_TDISCON_SUCCESSFUL : Word := 16#7011;   // status TDiscon called successfully
      SUB_STATUS_NO_ERROR : Word := 16#0000;   // NO error occured in subfunction call
      ERR_UNDEFINED_STATE : Word := 16#8600;   // Error: due to an undefined state in state machine
      ERR_IN_BLOCK_OPERATION : Word := 16#8001;   // Error: Wrong operation of the function block
      ERR_PARAMETRIZATION : Word := 16#8200;   // Error: during parameterization
      ERR_PROCESSING_EXTERN : Word := 16#8400;   // Error: when processing from outside (e. g. wrong I/O signals, axis not referenced)
      ERR_PROCESSING_INTERN : Word := 16#8600;   // Error: when processing internally (e. g. when calling a system function)
      ERR_AREA_RESERVED : Word := 16#8800;   // Error: Reserved area
      ERR_USER_DEFINED_CLASSES : Word := 16#9000;   // Error: User-defined error classes
      ERR_DISCONNECT : Word := 16#8601;   // Error: when calling tdiscon
      ERR_CONNECT : Word := 16#8602;   // Error: calling tcon
      ERR_PRELOGIN : Word := 16#8603;   // Error: executing prelogin
      ERR_PRELOGIN_DATA : Word := 16#8607;   // Error: converting prelogin data to word
      ERR_LOGIN : Word := 16#8604;   // Error: executing login
      ERR_LOGIN_DATA : Word := 16#8608;   // Error: converting login data to word
      ERR_TRCV : Word := 16#8605;   // Error: calling trcv
      ERR_ARCHIVE : Word := 16#8606;   // Error: archiving in db
      ERR_SQLBATCH_DATA : Word := 16#8609;   // Error: converting sql command data to word
      ERR_SQLBATCHSEND : Word := 16#8610;   // Error:sending sql data
   END_VAR
   // instTrcv.ADHOC := true;
BEGIN
   REGION BLOCK INFO HEADER
       //=============================================================================
       // Siemens AG (c)Copyright (2019)
       //-----------------------------------------------------------------------------
       // Library:       SQL
       // Target:        S7-1500 / FW 2.6
       // Engineering:   TIA Portal V15.1
       // Restrictions:  no
       // Requirements:  CPU 1500
       // Functionality: For database access:
       //                set up connection to SQL server, send batch and save answers from server
       //-----------------------------------------------------------------------------
       // Change log table:
       // Version    Date         Expert in charge           Changes applied
       // 01.00.00   30.05.2020   Siemens SUP Applications   First released version
       // 01.01.00   30.09.2020   Siemens SUP Applications   Added receiving of SQL database data
       //=============================================================================
   END_REGION

   #statEnable := #enable; // Work with temporary value / create process image

   REGION ENABLING/DISABLING
       IF (#statEnable = TRUE) AND (#statStatus = #STATUS_NO_CALL) THEN // Enable FB
           // First call; initialize FB
           #statValid := TRUE;
           #statBusy := TRUE;
           #statError := FALSE;
           #statErrorUserCleared := FALSE;
           #statErrorAutoCleared := FALSE;
           #statStatus := #STATUS_FIRST_CALL;
           #statSubfunctionStatus := #SUB_STATUS_NO_ERROR;
           #statFBErrorState := 0;
           #diagnostics := #statEmptyDiagnostics;
           #statDisablingCompleted := FALSE;
           #statSqlDataReceived := FALSE;

           // State machine - start functionality
           #statFBState := #FB_STATE_CONNECT;

           REGION Initialize functionality: call subsidiary FBs with FALSE
               #instTcon(REQ := FALSE,
                         ID := #connectionSettings.interfaceSettings.ID,
                         CONNECT := #connectionSettings.interfaceSettings);
               #instTrcv(EN_R := FALSE,
                         ID := #connectionSettings.interfaceSettings.ID,
                         DATA := #data.bytes);
               #instTdiscon(REQ := FALSE,
                            ID := #connectionSettings.interfaceSettings.ID);
               #instTsend(REQ := FALSE,
                          ID := #connectionSettings.interfaceSettings.ID,
                          LEN := DINT_TO_UINT(#statPreLoginLen),
                          DATA := #statPreLogin);
                               END_REGION

       ELSIF (#statEnable = FALSE) AND (#statEnableOld = TRUE) THEN // Disable FB 
           #statFBState := #FB_STATE_DISABLING;

       ELSIF (#statStatus = #STATUS_FIRST_CALL) THEN // Set status identifier of subsequent call
           #statStatus := #STATUS_SUBSEQUENT_CALL;
       END_IF;

       // Edge detection 'enable' input
       #statEnableOld := #statEnable;
   END_REGION ENABLING/DISABLING

   IF (#statStatus = #STATUS_NO_CALL) THEN // Nothing to do -> End here to reduce "system load"
       RETURN;
   END_IF;

   REGION STATE_MACHINE
       CASE #statFBState OF // State machine of FB
           #FB_STATE_NO_PROCESSING:
               REGION NO Processing
                   // No processing active (Note: this state must always be present and left empty)
                   ;
               END_REGION NO Processing

           #FB_STATE_INITIAL_DISCON:
               REGION make sure no connection is open before connecting          
                   #instTdiscon(REQ := TRUE,
                                ID := #connectionSettings.interfaceSettings.ID);

                   IF #instTdiscon.ERROR THEN
                       #statStatus := #ERR_DISCONNECT;
                       #statSubfunctionStatus := #instTdiscon.STATUS;
                       #statFBErrorState := #statFBState;
                       IF #ERR_TDISCON_REMOTE_TERMINATION = #instTdiscon.STATUS THEN
                           // disconnect done - proceed with wait for setup
                           // Error can be fixed by FB
                           #statStatus := #STATUS_TDISCON_SUCCESSFUL;
                           #instTdiscon(REQ := FALSE,
                                        ID := #connectionSettings.interfaceSettings.ID);
                           #statErrorAutoCleared := TRUE;
                           #statFBState := #FB_STATE_CONNECT;
                       ELSE
                           #statErrorUserCleared := TRUE;
                           #instTdiscon(REQ := FALSE,
                                        ID := #connectionSettings.interfaceSettings.ID);
                       END_IF;
                   ELSIF #instTdiscon.DONE THEN
                       #statStatus := #STATUS_TDISCON_SUCCESSFUL;
                       #instTdiscon(REQ := FALSE,
                                    ID := #connectionSettings.interfaceSettings.ID);
                       #statFBState := #FB_STATE_CONNECT;
                   END_IF;
               END_REGION ;

           #FB_STATE_CONNECT:
               REGION connecting
                   //if error was set in state before because of tdiscon error: #ERR_TDISCON_REMOTE_TERMINATION, reset
                   #statErrorAutoCleared := FALSE;

                   #instTcon(REQ := TRUE,
                             ID := #connectionSettings.interfaceSettings.ID,
                             CONNECT := #connectionSettings.interfaceSettings);

                   IF #instTcon.ERROR THEN
                       #statStatus := #ERR_CONNECT;
                       #statSubfunctionStatus := #instTcon.STATUS;
                       #statFBErrorState := #statFBState;
                       #statErrorUserCleared := TRUE;
                       #instTcon(REQ := FALSE,
                                 ID := #connectionSettings.interfaceSettings.ID,
                                 CONNECT := #connectionSettings.interfaceSettings);
                   ELSIF #instTcon.DONE THEN
                       #instTcon(REQ := FALSE,
                                 ID := #connectionSettings.interfaceSettings.ID,
                                 CONNECT := #connectionSettings.interfaceSettings);
                       #statFBState := #FB_STATE_PRELOGIN;
                   END_IF;
               END_REGION connecting

           #FB_STATE_PRELOGIN:
               REGION Prelogin active      
                   //copy data from data to cache
                   #statStatusPreLoginIntToWord := INT_TO_WORD(Serialize(SRC_VARIABLE := #statPreLoginData, DEST_ARRAY => #statPreLoginCache, POS := #tempPos));

                   IF #statStatusPreLoginIntToWord > 16#0000 THEN
                       #statStatus := #ERR_PRELOGIN_DATA;
                       #statSubfunctionStatus := #statStatusPreLoginIntToWord;
                       #statFBErrorState := #statFBState;
                       #statErrorUserCleared := TRUE;
                   END_IF;

                   //copy data from cache to preLogin (without unwanted filled zero bytes)
                   FOR #tempCounter := 0 TO #tempPos DO
                       //when serializing prelogin data a zero is added in between types
                       //delete these zeros
                       CASE #tempCounter OF
                           9, 15, 21, 27, 33, 39, 45, 51:
                               #tempGaps += 1;
                           ELSE
                               #statPreLogin[#tempCounter - #tempGaps] := #statPreLoginCache[#tempCounter];
                       END_CASE;

                   END_FOR;

                   //write number of bytes, that have to be transmitted, to preLoginLen (adjusted by the deleted gaps)
                   #statPreLoginLen := #tempPos - #tempGaps;

                   #instTsend(REQ := TRUE,
                              ID := #connectionSettings.interfaceSettings.ID,
                              LEN := DINT_TO_UINT(#statPreLoginLen),
                              DATA := #statPreLogin);

                   IF #instTsend.ERROR THEN
                       #statStatus := #ERR_PRELOGIN;
                       #statErrorUserCleared := TRUE;
                       #statSubfunctionStatus := #instTsend.STATUS;
                       #statFBErrorState := #statFBState;
                       #instTsend(REQ := FALSE,
                                  ID := #connectionSettings.interfaceSettings.ID,
                                  DATA := #statPreLogin);

                   ELSIF #instTsend.DONE THEN
                       #instTsend(REQ := FALSE,
                                  ID := #connectionSettings.interfaceSettings.ID,
                                  DATA := #statPreLogin);
                       #statFBState := #FB_STATE_LOGIN;
                   END_IF;

               END_REGION Prelogin

           #FB_STATE_LOGIN: // Login active
               REGION Login
                   REGION write login data to DB
                       #statWriter := 0; //varible for iterating through data array
                       #tempPos := 0;

                       REGION write String TO data AND set length AND offset in offsetLength (hostName)
                           "LSql_WriteData"(inString := #connectionSettings.loginInformation.hostName,
                                          offsetOwn := #statLoginData.login.offsetLength.hostName.offset,
                                          offsetNext => #statLoginData.login.offsetLength.userName.offset,
                                          length => #statLoginData.login.offsetLength.hostName.length,
                                          error => #statErrorWriteData,
                                          status => #statWriteData,
                                          data := #statLoginData.login.data,
                                          writer := #statWriter);

                           //write string to data and set length and offset in offsetLength (userName)
                         "LSql_WriteData"(inString := #connectionSettings.loginInformation.userName,
                                          offsetOwn := #statLoginData.login.offsetLength.userName.offset,
                                          offsetNext => #statLoginData.login.offsetLength.password.offset,
                                          length => #statLoginData.login.offsetLength.userName.length,
                                          error => #statErrorWriteData,
                                          status => #statWriteData,
                                          data := #statLoginData.login.data,
                                          writer := #statWriter);

                           //write string to data and set length and offset in offsetLength (password)
                         "LSql_WritePassword"(inString := #connectionSettings.loginInformation.password,
                                              offsetOwn := #statLoginData.login.offsetLength.password.offset,
                                              offsetNext => #statLoginData.login.offsetLength.appName.offset,
                                              length => #statLoginData.login.offsetLength.password.length,
                                              error => #statErrorWriteData,
                                              status => #statWriteData,
                                              data := #statLoginData.login.data,
                                              writer := #statWriter);

                           //write string to data and set length and offset in offsetLength (appName)
                         "LSql_WriteData"(inString := #connectionSettings.loginInformation.appName,
                                          offsetOwn := #statLoginData.login.offsetLength.appName.offset,
                                          offsetNext => #statLoginData.login.offsetLength.serverName.offset,
                                          length => #statLoginData.login.offsetLength.appName.length,
                                          error => #statErrorWriteData,
                                          status => #statWriteData,
                                          data := #statLoginData.login.data,
                                          writer := #statWriter);

                           //write string to data and set length and offset in offsetLength (serverName)
                         "LSql_WriteData"(inString := #connectionSettings.loginInformation.serverName,
                                          offsetOwn := #statLoginData.login.offsetLength.serverName.offset,
                                          offsetNext => #statLoginData.login.offsetLength.unused.offset,
                                          length => #statLoginData.login.offsetLength.serverName.length,
                                          error => #statErrorWriteData,
                                          status => #statWriteData,
                                          data := #statLoginData.login.data,
                                          writer := #statWriter);

                           //write string to data and set length and offset in offsetLength (unused)
                           "LSql_WriteData"(inString := '',
                                          offsetOwn := #statLoginData.login.offsetLength.unused.offset,
                                          offsetNext => #statLoginData.login.offsetLength.libraryName.offset,
                                          length => #statLoginData.login.offsetLength.unused.length,
                                          error => #statErrorWriteData,
                                          status => #statWriteData,
                                          data := #statLoginData.login.data,
                                          writer := #statWriter);

                           //write string to data and set length and offset in offsetLength (libraryName)
                         "LSql_WriteData"(inString := #connectionSettings.loginInformation.libraryName,
                                          offsetOwn := #statLoginData.login.offsetLength.libraryName.offset,
                                          offsetNext => #statLoginData.login.offsetLength.local.offset,
                                          length => #statLoginData.login.offsetLength.libraryName.length,
                                          error => #statErrorWriteData,
                                          status => #statWriteData,
                                          data := #statLoginData.login.data,
                                          writer := #statWriter);

                           //wrtie string to data and set length and offset in offsetLength (local)
                         "LSql_WriteData"(inString := #connectionSettings.loginInformation.local,
                                          offsetOwn := #statLoginData.login.offsetLength.local.offset,
                                          offsetNext => #statLoginData.login.offsetLength.databaseName.offset,
                                          length => #statLoginData.login.offsetLength.local.length,
                                          error => #statErrorWriteData,
                                          status => #statWriteData,
                                          data := #statLoginData.login.data,
                                          writer := #statWriter);

                           //write string to data and set length and offset in offsetLength (databaseName)
                         "LSql_WriteData"(inString := #connectionSettings.loginInformation.databaseName,
                                          offsetOwn := #statLoginData.login.offsetLength.databaseName.offset,
                                          offsetNext => #statLoginData.login.offsetLength.sspi.offset,
                                          length => #statLoginData.login.offsetLength.databaseName.length,
                                          error => #statErrorWriteData,
                                          status => #statWriteData,
                                          data := #statLoginData.login.data,
                                          writer := #statWriter);

                           //string string to data and set length and offset in offsetLength (sspi)
                         "LSql_WriteData"(inString := #connectionSettings.loginInformation.sspi,
                                          offsetOwn := #statLoginData.login.offsetLength.sspi.offset,
                                          offsetNext => #statLoginData.login.offsetLength.atchDbFile.offset,
                                          length => #statLoginData.login.offsetLength.sspi.length,
                                          error => #statErrorWriteData,
                                          status => #statWriteData,
                                          data := #statLoginData.login.data,
                                          writer := #statWriter);

                           //string to data and set length and offset in offsetLength (atchDbFile)
                         "LSql_WriteData"(inString := #connectionSettings.loginInformation.attachDbfile,
                                          offsetOwn := #statLoginData.login.offsetLength.atchDbFile.offset,
                                          offsetNext => #statLoginData.login.offsetLength.changePassword.offset,
                                          length => #statLoginData.login.offsetLength.atchDbFile.length,
                                          error => #statErrorWriteData,
                                          status => #statWriteData,
                                          data := #statLoginData.login.data,
                                          writer := #statWriter);

                           //string to data and set length and offset in offsetLength (changePassword)
                         "LSql_WritePassword"(inString := #connectionSettings.loginInformation.changePassword,
                                              offsetOwn := #statLoginData.login.offsetLength.changePassword.offset,
                                              offsetNext => #statLoginData.login.length,
                                              length => #statLoginData.login.offsetLength.changePassword.length,
                                              error => #statErrorWriteData,
                                              status => #statWriteData,
                                              data := #statLoginData.login.data,
                                              writer := #statWriter);
                       END_REGION ;

                       //set length parameters according to added data
                       #tempLengthAsInt := DWORD_TO_DINT(#statLoginData.login.length);
                       //rotate by 8 because word
                       #tempLengthRor := ROR(IN := #tempLengthAsInt, N := 8) + 8;
                       #statLoginData.header.length := DINT_TO_WORD( #tempLengthRor);

                       //shift by 16 dword
                       #statLoginData.login.length := SHL(IN := #statLoginData.login.length, N := 16);

                   END_REGION

                   //copy standard data to login
                   #statStatusLoginIntToWord := INT_TO_WORD(Serialize(SRC_VARIABLE := #statLoginData, DEST_ARRAY => #statLogin, POS := #tempPos));
                   //check for error in INT_TO_WORD
                   IF #statStatusLoginIntToWord > 16#0000 THEN
                       #statStatus := #ERR_LOGIN_DATA;
                       #statSubfunctionStatus := #statStatusLoginIntToWord;
                       #statFBErrorState := #statFBState;
                       #statErrorUserCleared := TRUE;
                   END_IF;

                   //write length to loginLen (adjusted by the length of the data (-1024+writer) and deleted gaps in the header)
                   #statLoginLen := #tempPos - 1024 + #statWriter;
                   // BG TODO - warum 1024 - nicht 2048?
                   // Keine magic numbers ;)

                   //deletes last zero byte, if necessary
                   // BG TODO ein kommentar dazu der aussagt warum modulo 2 addiert wird wäre dann antürlich notwendig
                   #statLoginLen := #statLoginLen + #tempPos MOD 2;

                   #statFBState := #FB_STATE_SENDLOGIN;
               END_REGION ; 

           #FB_STATE_SENDLOGIN:
               REGION send login data
                   #instTsend(REQ := #enable,
                              ID := #connectionSettings.interfaceSettings.ID,
                              LEN := DINT_TO_UINT(#statLoginLen),
                              DATA := #statLogin);

                   IF #instTsend.ERROR THEN
                       #statStatus := #ERR_LOGIN;
                       #statSubfunctionStatus := #instTsend.STATUS;
                       #statFBErrorState := #statFBState;
                       #statErrorUserCleared := TRUE;
                       #instTsend(REQ := FALSE,
                                  ID := #connectionSettings.interfaceSettings.ID,
                                  DATA := #statLogin);
                   ELSIF #instTsend.DONE THEN
                       #instTsend(REQ := FALSE,
                                  ID := #connectionSettings.interfaceSettings.ID,
                                  DATA := #statLogin);
                       #statFBState := #FB_STATE_SQLBATCH;
                   END_IF;
                   // TBD: after sending is complete, receiving and evaluating the content is necessary to switch to the next state!
               END_REGION send login data

           #FB_STATE_SQLBATCH:
               REGION sqlbatch execution
                   REGION receive data
                       #instTrcv(EN_R := TRUE,
                                 ID := #connectionSettings.interfaceSettings.ID,
                                 DATA := #data.bytes,
                                 RCVD_LEN => #statReceivedBytes);
                       //TRCV DATA in previous version V1.0.0: #statReceiveBuffer as Array[0..1023] of Byte, followed by deserialize
                       IF #instTrcv.NDR THEN
                           #statSqlDataReceived := TRUE;
                           // #statDeserializeStatus := Deserialize(SRC_ARRAY := #statReceiveBuffer, DEST_VARIABLE =>#SqlReceiveData, POS := #statDeserializePosition);
                           // Clear the statReceiveBuffer
                           // FILL_BLK(IN:=16#00,
                           //          COUNT:=#statReceivedBytes,
                           //          OUT=>#statReceiveBuffer.bytes[0]);
                           // #statReceivedBytes := 0;
                       ELSE
                           #statSqlDataReceived := FALSE;
                       END_IF;

                       IF #instTrcv.ERROR THEN
                           #statStatus := #ERR_TRCV;
                           #statErrorUserCleared := TRUE;
                           #statSubfunctionStatus := #instTrcv.STATUS;
                           #statFBErrorState := #statFBState;
                       END_IF;
                   END_REGION receive data


                   REGION send sql command
                       //get positive edge of executeSqlBatch
                       IF #executeCommand AND NOT #statExecuteSqlBatchOld THEN

                           #statWriter := 0;

                           //write string to data and set length parameter accoding to the added data
                           "LSql_WriteData"(inString := #command,
                                            offsetOwn := 16#1E00,
                                            offsetNext => #statSqlBatchData.header.length,
                                            error => #statErrorWriteData,
                                            status => #statWriteData,
                                            length => #tempLength,
                                            data := #statSqlBatchData.sqlBatch.sqlText,
                                            writer := #statWriter);

                           //transform (lowByte highByte) to (highByte lowByte)
                           #statSqlBatchData.header.length := ROR(IN := #statSqlBatchData.header.length, N := 8);

                           //copy data from data to cache
                           #statStatusSqlBatchIntToWord := INT_TO_WORD(Serialize(SRC_VARIABLE := #statSqlBatchData, DEST_ARRAY => #statSqlBatch, POS := #tempPos));
                           //check for error in Int_To_Word Function
                           IF #statStatusSqlBatchIntToWord > 16#0000 THEN
                               #statStatus := #ERR_SQLBATCH_DATA;
                               #statSubfunctionStatus := #statStatusSqlBatchIntToWord;
                               #statFBErrorState := #statFBState;
                               #statErrorUserCleared := TRUE;
                           END_IF;
                           //write length to DB, adjusted by the length of the data (-1024+writer)
                           #statSqlBatchLen := #tempPos - 1024 + #statWriter;

                           //deletes last zero byte, if necessary

                           #statSqlBatchLen += #tempPos MOD 2;
                           #statTransmissionSqlCommand := TRUE;
                           #statExecuteSqlBatchOld := #executeCommand;
                       END_IF; //finished creating stream 

                       //get the negative edge 
                       IF NOT #executeCommand AND #statExecuteSqlBatchOld THEN
                           #statExecuteSqlBatchOld := #executeCommand;
                       END_IF;

                       //send data
                       IF #statTransmissionSqlCommand THEN
                           #instTsend(REQ := TRUE,
                                      ID := #connectionSettings.interfaceSettings.ID,
                                      LEN := DINT_TO_UINT(#statSqlBatchLen),
                                      DATA := #statSqlBatch);
                           //check for error in Tsend
                           IF #instTsend.ERROR THEN
                               #statStatus := #ERR_SQLBATCHSEND;
                               #statSubfunctionStatus := #instTsend.STATUS;
                               #statFBErrorState := #statFBState;
                               #statErrorUserCleared := TRUE;
                               #statTransmissionSqlCommand := FALSE;
                           ELSIF #instTsend.DONE THEN
                               #instTsend(REQ := FALSE,
                                          ID := #connectionSettings.interfaceSettings.ID,
                                          LEN := DINT_TO_UINT(#statSqlBatchLen),
                                          DATA := #statSqlBatch);
                               #statTransmissionSqlCommand := FALSE;
                           END_IF;
                       END_IF;

                   END_REGION send sql command

               END_REGION sqlbatch execution

           #FB_STATE_DISABLING: // Disconnect active
               REGION Disabling
                   #instTrcv(EN_R := FALSE,
                             ID := #connectionSettings.interfaceSettings.ID,
                             DATA := #data.bytes);
               END_REGION
               REGION Disconnect
                   //disconnect function, closes the connection to the server
                   #instTdiscon(REQ := TRUE,
                                ID := #connectionSettings.interfaceSettings.ID);

                   IF #instTdiscon.ERROR THEN
                       #statStatus := #ERR_DISCONNECT;
                       #statSubfunctionStatus := #instTdiscon.STATUS;
                       #statFBErrorState := #statFBState;
                       IF #ERR_TDISCON_REMOTE_TERMINATION = #instTdiscon.STATUS THEN
                           #statDisablingCompleted := TRUE;

                           #instTdiscon(REQ := FALSE,
                                        ID := #connectionSettings.interfaceSettings.ID);
                       ELSE

                           #statErrorUserCleared := TRUE;
                           #instTdiscon(REQ := FALSE,
                                        ID := #connectionSettings.interfaceSettings.ID);
                       END_IF;

                   ELSIF #instTdiscon.DONE THEN
                       //#statSqlConnectionEstablished := FALSE;
                       #instTdiscon(REQ := FALSE,
                                    ID := #connectionSettings.interfaceSettings.ID);
                   END_IF;
                   #statFBState := #FB_STATE_NO_PROCESSING;


                   #statDisablingCompleted := TRUE;
               END_REGION Disconnect


           ELSE // Undefined state in state machine reached
               REGION undefined state        
                   #statStatus := #ERR_UNDEFINED_STATE;
                   #statErrorUserCleared := TRUE;
               END_REGION undefined state
       END_CASE;
   END_REGION STATE_MACHINE

   REGION OUTPUTS
       // Write outputs
       IF (#statDisablingCompleted = TRUE) THEN
           REGION disabling
               // Reset outputs if disabling completed
               #statValid := FALSE;
               #statBusy := FALSE;
               #statError := FALSE;
               #statErrorUserCleared := FALSE;
               #statErrorAutoCleared := FALSE;
               #statStatus := #STATUS_NO_CALL;

           END_REGION disabling

       ELSIF (#statErrorUserCleared = TRUE) AND (#statError = FALSE) THEN
           REGION error user cleared
               // Error can only be cleared by user; rising edge at enable input is needed to continue 
               #statValid := FALSE;
               #statBusy := FALSE;
               #statError := TRUE;
               // Write diagnostics
               #diagnostics.status := #statStatus;
               #diagnostics.subfunctionStatus := #statSubfunctionStatus;
               #diagnostics.stateNumber := #statFBErrorState;
               // execution aborted --> set state no processing
               #statFBState := #FB_STATE_NO_PROCESSING;
           END_REGION error user cleared

       ELSIF (#statErrorAutoCleared = TRUE) AND (#statError = FALSE) THEN
           REGION error auto cleared
               // Error can be reset by FB automatically
               #statValid := FALSE;
               #statBusy := TRUE;
               #statError := TRUE;
               // Write diagnostics
               #diagnostics.status := #statStatus;
               #diagnostics.subfunctionStatus := #statSubfunctionStatus;
               #diagnostics.stateNumber := #statFBErrorState;
           END_REGION error auto cleared

       ELSIF (#statErrorAutoCleared = FALSE) AND (#statErrorUserCleared = FALSE) AND (#statError = TRUE) THEN
           REGION after user/auto cleared
               // If autocleared error is acknowledged
               #statValid := TRUE;
               #statBusy := TRUE;
               #statError := FALSE;
               // TODO: remove this line if more detailed status information is used instead of "#STATUS_SUBSEQUENT_CALL"
               #statStatus := #STATUS_SUBSEQUENT_CALL;
           END_REGION after user/auto cleared
       END_IF;

       REGION Write static values to outputs
           #valid := #statValid;
           #busy := #statBusy;
           #error := #statError;
           #status := #statStatus;
           #dataReceived := #statSqlDataReceived;
           // if ENO mechanism is not used / not wanted replace the following line by --> ENO := TRUE;
           ENO := NOT #statError;

       END_REGION Write static values to outputs
   END_REGION OUTPUTS
END_FUNCTION_BLOCK

// folder: LSql/Helpers

FUNCTION "LSql_WriteData" : Void   // FC4, SCL
{ S7_Optimized_Access := 'TRUE' }
VERSION : 0.1
   VAR_INPUT
      inString : String;   // string to insert
      offsetOwn : Word;   // offset of the string
   END_VAR
   VAR_OUTPUT
      error : Bool;   // TRUE: An error occurred during the execution of the FC
      status : Word;   // 16#0000 - 16#7FFF: Status of the FB, 16#8000 - 16#FFFF: Error identification
      offsetNext : Word;   // offset of the next string
      length : Word;   // length of the string after conversion
   END_VAR
   VAR_IN_OUT
      data : Array[0..1023] of Byte;   // array where string should be inserted
      writer : Int;   // number of the element to be written
   END_VAR
   VAR_TEMP
      tempStatus : Word;   // temp value for output 'status'
      tempBytes : Array[0..1023] of Byte;   // temp for char array after conversion
      tempLen : DInt;   // length of data before filling in zero bytes
      tempCounter : DInt;   // counter for loop to go through data
      tempOffsetNext : Word;   // offset of converted data, added up to input offset
      tempLength : Word;   // length of data
      tempOffsetAsDInt : DInt;   // offset as a dint
      tempLenAsUInt : UInt;   // length as uint
   END_VAR
   VAR CONSTANT
      STATUS_FINISHED_NO_ERROR : Word := 16#0000;   // NO error - execution finished without errors
      ERR_UNDEFINED : Word := 16#8000;   // Error: due to an undefined case
      ERR_IN_BLOCK_OPERATION : Word := 16#8001;   // Error: Wrong operation of the function block
      ERR_PARAMETRIZATION : Word := 16#8200;   // Error: during parameterization
      ERR_PROCESSING_EXTERN : Word := 16#8400;   // Error: when processing from outside (e. g. wrong I/O signals, axis not referenced)
      ERR_PROCESSING_INTERN : Word := 16#8600;   // Error: when processing internally (e. g. when calling a system function)
      ERR_AREA_RESERVED : Word := 16#8800;   // Error: Reserved area
      ERR_USER_DEFINED_CLASSES : Word := 16#9000;   // Error: User-defined error classes
   END_VAR
BEGIN
   REGION BLOCK INFO HEADER
       //===============================================================================
       // (Siemens AG (c)Copyright (2020)
       //-------------------------------------------------------------------------------
       // Title:            LSql_WriteData
       // Comment/Function: serialize input string to array of bytes
       // Library/Family:   LSql
       // Author:           Siemens SUP Applications 
       //Target:            S7-1500 / FW 2.6
       // Engineering:      TIA Portal (V16)
       // Restrictions:     no
       // Requirements:      CPU 1500
       //-------------------------------------------------------------------------------
       // Change log table:
       // Version  | Date       | Expert in charge         | Changes applied
       //----------|------------|--------------------------|------------------------------
       // 01.00.00 | 2020-02-19 | Siemens SUP Applications | First released version
       //===============================================================================
   END_REGION

   REGION INITIALISATION  
       // TODO: Initialize functionality: reset of variables, diagnostics, etc.
       #tempLenAsUInt := 0;
       #tempLen := 0;
       #tempCounter := 0;
       #tempOffsetAsDInt := 0;
       #tempOffsetNext := 16#0000;
       #tempStatus := #STATUS_FINISHED_NO_ERROR;
   END_REGION

   REGION PROGRAM LOGIC
       //convert string to char array
       Strg_TO_Chars(Strg := #inString,
                     pChars := 0,
                     Cnt => #tempLenAsUInt,
                     Chars := #tempBytes);
       #tempLen := UINT_TO_DINT(#tempLenAsUInt);


       //fill in zero bytes between each letter
       FOR #tempCounter := 0 TO #tempLen - 1 DO
           #data[#writer] := #tempBytes[#tempCounter];
           #writer += 1;
           #data[#writer] := 16#00;
           #writer += 1;
       END_FOR;


       //set offset to length * 2 cause of filled in zero bytes
       #tempOffsetAsDInt := WORD_TO_DINT(#offsetOwn);
       #tempOffsetAsDInt := ROR(IN := #tempOffsetAsDInt, N := 8) + #tempLen * 2;
       #tempOffsetNext := DINT_TO_WORD(#tempOffsetAsDInt);
       #tempOffsetNext := ROL(IN := #tempOffsetNext, N := 8);


       //set length to the number of letters(low Byte, high Byte)
       #tempLength := ROL(IN := DINT_TO_WORD(#tempLen), N := 8);
       // so lassen

   END_REGION

   REGION OUTPUTS

       #offsetNext := #tempOffsetNext;
       #length := #tempLength;
       #error := #tempStatus.%X15;
       #status := #tempStatus;
       // if ENO mechanism is not used / not wanted replace the following line by --> ENO := TRUE;
       ENO := NOT #tempStatus.%X15;
   END_REGION
END_FUNCTION

FUNCTION "LSql_WritePassword" : Void   // FC5, SCL
{ S7_Optimized_Access := 'TRUE' }
VERSION : 0.1
   VAR_INPUT
      inString : String;   // string to be inserted
      offsetOwn : Word;   // offset of the current string
   END_VAR
   VAR_OUTPUT
      error : Bool;   // TRUE: An error occurred during the execution of the FC
      status : Word;   // 16#0000 - 16#7FFF: Status of the FB, 16#8000 - 16#FFFF: Error identification
      offsetNext : Word;   // offset of the next string
      length : Word;   // length of the string after conversion
   END_VAR
   VAR_IN_OUT
      data : Array[0..1023] of Byte;   // array where string should be inserted
      writer : Int;   // number of the next element that should be written
   END_VAR
   VAR_TEMP
      tempStatus : Word;   // temp value for output 'status'
      tempConvBytes : Array[0..123] of Byte;   // converted bytes
      tempLen : DInt;   // length of data after conversion to char array
      tempCounter : DInt;   // variable for loop to go through data
      tempLenAsUInt : UInt;   // length as uint
      tempOffsetNext : Word;   // offset of data for output, added to input offset
      tempOffsetAsDInt : DInt;   // offset as dint
      tempLength : Word;   // length of data
   END_VAR
   VAR CONSTANT
      STATUS_FINISHED_NO_ERROR : Word := 16#0000;   // NO error - execution finished without errors
      ERR_UNDEFINED : Word := 16#8000;   // Error: due to an undefined case
      ERR_IN_BLOCK_OPERATION : Word := 16#8001;   // Error: Wrong operation of the function block
      ERR_PARAMETRIZATION : Word := 16#8200;   // Error: during parameterization
      ERR_PROCESSING_EXTERN : Word := 16#8400;   // Error: when processing from outside (e. g. wrong I/O signals, axis not referenced)
      ERR_PROCESSING_INTERN : Word := 16#8600;   // Error: when processing internally (e. g. when calling a system function)
      ERR_AREA_RESERVED : Word := 16#8800;   // Error: Reserved area
      ERR_USER_DEFINED_CLASSES : Word := 16#9000;   // Error: User-defined error classes
   END_VAR
BEGIN
   REGION BLOCK INFO HEADER
       //===============================================================================
       // (Siemens AG (c)Copyright (2020)
       //-------------------------------------------------------------------------------
       // Title:            LSql_WriteData
       // Comment/Function: serialize input string (password) to array of bytes
       // Library/Family:   LSql
       // Author:           Siemens SUP Applications 
       //Target:            S7-1500 / FW 2.6
       // Engineering:      TIA Portal (V16)
       // Restrictions:     no
       // Requirements:      CPU 1500
       //-------------------------------------------------------------------------------
       // Change log table:
       // Version  | Date       | Expert in charge         | Changes applied
       //----------|------------|--------------------------|------------------------------
       // 01.00.00 | 2020-02-19 | Siemens SUP Applications | First released version
       //===============================================================================
   END_REGION

   REGION INITIALISATION  
       // TODO: Initialize functionality: reset of variables, diagnostics, etc.
       #tempLenAsUInt := 0;
       #tempLen := 0;
       #tempCounter := 0;
       #tempOffsetAsDInt := 0;
       #tempOffsetNext := 16#0000;
       #tempStatus := #STATUS_FINISHED_NO_ERROR;
   END_REGION

   REGION PROGRAM LOGIC
       Strg_TO_Chars(Strg := #inString,
                     pChars := 0,
                     Cnt => #tempLenAsUInt,
                     Chars := #tempConvBytes);
       #tempLen := UINT_TO_DINT(#tempLenAsUInt);

       //convert password (switch low<->high bits and xor 16#A5)
       FOR #tempCounter := 0 TO #tempLen - 1 DO
           #tempConvBytes[#tempCounter] := ROR(IN := #tempConvBytes[#tempCounter], N := 4) XOR 16#A5;
       END_FOR;

       //fill in 16#A5 bytes between each letter
       FOR #tempCounter := 0 TO #tempLen - 1 DO
           #data[#writer] := #tempConvBytes[#tempCounter];
           #writer += 1;
           #data[#writer] := 16#A5;
           #writer += 1;
       END_FOR;

       //set offset to length * 2 cause of filled in zero bytes
       #tempOffsetAsDInt := WORD_TO_DINT(#offsetOwn);
       #tempOffsetAsDInt := ROR(IN := #tempOffsetAsDInt, N := 8) + #tempLen * 2;
       #tempOffsetNext := DINT_TO_WORD(#tempOffsetAsDInt);
       #tempOffsetNext := ROL(IN := #tempOffsetNext, N := 8);

       //set length to the number of letters(low Byte, high Byte)
       #tempLength := ROL(IN := DINT_TO_WORD(#tempLen), N := 8);
   END_REGION

   REGION OUTPUTS
       #length := #tempLength;
       #offsetNext := #tempOffsetNext;
       #error := #tempStatus.%X15;
       #status := #tempStatus;
       // if ENO mechanism is not used / not wanted replace the following line by --> ENO := TRUE;
       ENO := NOT #tempStatus.%X15;
   END_REGION
END_FUNCTION

// ===== library types =====

TYPE "LSql_typeReceivedData"
   STRUCT
      len : UDInt;   // number of bytes received / number of bytes contained in message
      bytes : Array[0..1023] of Byte;   // space for receiving data / recieved message
   END_STRUCT;
END_TYPE

TYPE "LSql_typeTokenRow"
   STRUCT
      length : Byte;
      data : DWord;
   END_STRUCT;
END_TYPE